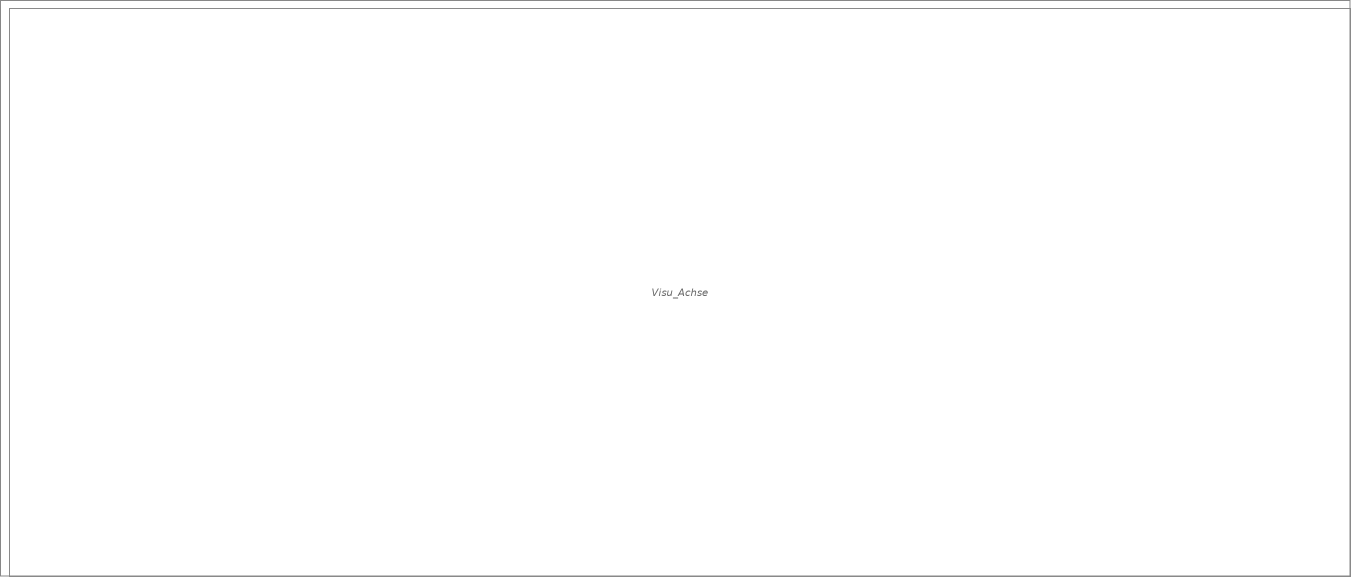
VISUALIZATION Achse_T  // 1351x577
    Frame (9,8 1342x569)
        shows Visu_Achse(Axis := MAIN.Axis_T)
END_VISUALIZATION

(* stored: Version 1.1.0.1, ProductVersion 3.1.4024.10
   Visu Achse_T: Id {35b28d0c-ceeb-4501-9f7a-b33cf5763810} *)
